ABB RobotStudio station: Projet3_V1_Robot.rsstn

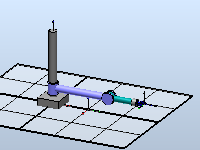
Station Lab3_2e_Robot (saved by RobotStudio format 3)
Layout (positions relative to the parent item):
  - My_Mechanism [mechanism] at (0, 0, 0) mm; joint values [0, 0, 0, 0] (rad or m)
      links: L1, L2, L3, L4, L5
  - MyPince [mechanism] at (0, 0, 0) mm
      TCP MyPince at (315, 0, 1200) mm, rotated rx 180 ry 0 rz 180 deg
      links: pince
  - Atelier [graphiccomponentgroup] at (-500, 0, 0) mm, rotated rx 0 ry 0 rz 180 deg
    - fleche_droite [part]
    - fleche_droite_2_2 [part] at (0, 0, 0) mm, rotated rx 90 ry 0 rz 90 deg
    - fleche_droite_2 [part] at (0, 0, 0) mm, rotated rx 90 ry 0 rz 0 deg
    - Objet_1 [part]
  - F0 [graphiccomponentgroup] at (0, 0, 0) mm, rotated rx 0 ry 0 rz -90 deg
    - fleche_droite [part] at (0, 0, 963.46) mm
    - fleche_droite_2_2 [part] at (71.94, 0, 0) mm, rotated rx 90 ry 0 rz 90 deg
    - fleche_droite_2 [part] at (0, -76.42, 0) mm, rotated rx 90 ry 0 rz 0 deg
    - Objet_1 [part]
  - Outil [graphiccomponentgroup] at (-1300, 0, 215) mm, rotated rx -90 ry 0 rz 90 deg
    - fleche_droite [part]
    - fleche_droite_2_2 [part] at (0, 0, 0) mm, rotated rx 90 ry 0 rz 90 deg
    - fleche_droite_2 [part] at (0, 0, 0) mm, rotated rx 90 ry 0 rz 0 deg
    - Objet_1 [part]
  - Wobj0 [frame] at (-500, 0, 0) mm, rotated rx 0 ry 0 rz 90 deg
  - RepereOutil [frame] at (-1300, 0, 215) mm, rotated rx 0 ry -90 rz 0 deg
Attachment: MyPince is attached to My_Mechanism / L5
Attachment: RepereOutil is attached to MyPince / pince
Attachment: Outil is attached to MyPince / pince
Targets, tools, work objects and paths stored in the station, written as RAPID:
! task (no controller)
MODULE CalibData
  PERS tooldata MyPince:=[TRUE,[[0,0,100],[1,0,0,0]],[1,[1,0,0],[1,0,0,0],0,0,0]];
ENDMODULE

